FUNCTION AcCheck : BOOL
VAR_INPUT
	r_Voltage	: REAL;
	r_Frequency	: REAL;
END_VAR

AcCheck	:= AcFrequencyCheck(r_Frequency) AND AcVoltageCheck(r_Voltage);

END_FUNCTION

(* stored: Version 1.1.0.1, ProductVersion 3.1.4026.18
   POU AcCheck: Id {dd403a1c-6e52-4e29-9d55-43f2ac623397}, SpecialFunc None *)
